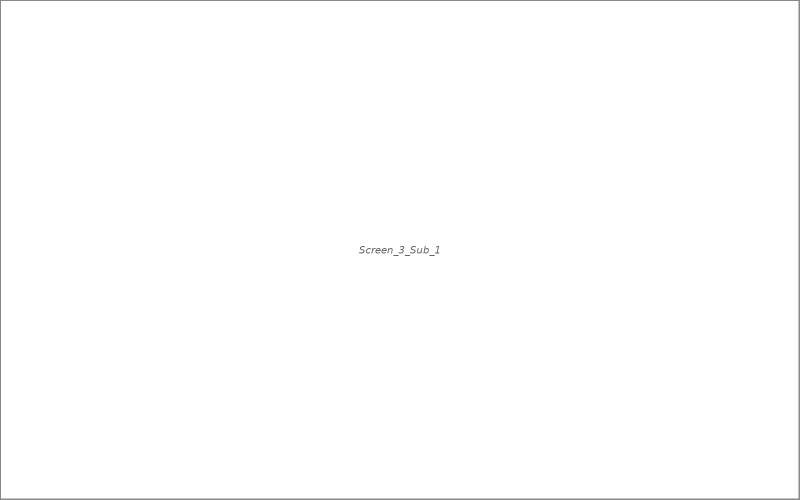
VISUALIZATION Screen_3  // 800x500
    TabControl (0,0 800x500), frame switch variable: GVL.HMI_Heading[2]
        shows Screen_3_Sub_1()
        [0]: TabTitle=Maintenance
END_VISUALIZATION

(* stored: Version 1.1.0.1, ProductVersion 3.1.4024.12
   Visu Screen_3: Id {fa18eb08-88b8-4fde-92ee-b970344cdc05} *)
